Staubli VAL3: SplitJoint.pgx

public program SplitJoint(string x_sSLine, string x_sTitle, jointRx& x_jJ, bool& x_bRes)
  local trsf l_trTrsf
  local num l_nData[6]
  local string l_sChar[2]
begin

//  call SplitTrsf(x_sSLine,x_sTitle,l_trTrsf,x_bRes)
//  if x_bRes
//    x_jJ.j1=l_trTrsf.x
//    x_jJ.j2=l_trTrsf.y
//    x_jJ.j3=l_trTrsf.z
//    x_jJ.j4=l_trTrsf.rx
//    x_jJ.j5=l_trTrsf.ry
//    x_jJ.j6=l_trTrsf.rz
//
//  endIf


  x_bRes=false

  if x_sSLine==""
    return
  endIf

  x_sSLine=right(x_sSLine,len(x_sSLine)-len(x_sTitle))

  //解析每一行
  l_sChar[0]=","
  l_sChar[1]=","

  call SplitNumS(x_sSLine,l_nData,l_sChar,x_bRes)

  if !x_bRes
    return
  endIf

  x_jJ.j1=l_nData[0]
  x_jJ.j2=l_nData[1]
  x_jJ.j3=l_nData[2]
  x_jJ.j4=l_nData[3]
  x_jJ.j5=l_nData[4]
  x_jJ.j6=l_nData[5]






end
